// TIA Portal V15.1 export
// export: Created 2024-05-17T05:38:09.4997729Z, ExportSetting WithDefaults, DisplayName Totally Integrated Automation Portal, DisplayVersion V15.1 Update 5, DisplayName TIA Portal Openness, DisplayVersion V15.1 Update 5, DisplayName SINAMICS Startdrive Advanced, DisplayVersion V15.1, DisplayName G130, G150, S120, S150, SINAMICS MV, S210, DisplayVersion V15.1, DisplayName G110M, G120, G120C, G120D, G120P, DisplayVersion V15.1, DisplayName STEP 7 Professional, DisplayVersion V15.1 Update 5, DisplayName STEP 7 Safety, DisplayVersion V15.1, DisplayName WinCC Professional, DisplayVersion V15.1 Update 5, DisplayName SIMATIC Visualization Architect, DisplayVersion V15.1
ORGANIZATION_BLOCK "209000NCP01"   // OB1, FBD, ProgramCycle
TITLE = 209000NCP01
{ S7_Optimized_Access := 'FALSE' }
VERSION : 0.1
// stored: AutoNumber false, IsIECCheckEnabled false, SetENOAutomatically False
   VAR_TEMP
      OB1_EV_CLASS : Byte;   // Bits 0-3 = 1 (Coming event), Bits 4-7 = 1 (Event class 1)
      OB1_SCAN_1 : Byte;   // 1 (Cold restart scan 1 of OB 1), 3 (Scan 2-n of OB 1)
      OB1_PRIORITY : Byte;   // Priority of OB Execution
      OB1_OB_NUMBR : Byte;   // 1 (Organization block 1, OB1)
      OB1_RESERVED_1 : Byte;   // Reserved for system
      OB1_RESERVED_2 : Byte;   // Reserved for system
      OB1_PREV_CYCLE : Int;   // Cycle time of previous OB1 scan (milliseconds)
      OB1_MIN_CYCLE : Int;   // Minimum cycle time of OB1 (milliseconds)
      OB1_MAX_CYCLE : Int;   // Maximum cycle time of OB1 (milliseconds)
      OB1_DATE_TIME : Date_And_Time;   // Date and time OB1 started
   END_VAR
BEGIN

REGION Network 1: **** 1 - Inputs **** Incrementation of number of executions
   // Incrementation of number of executions
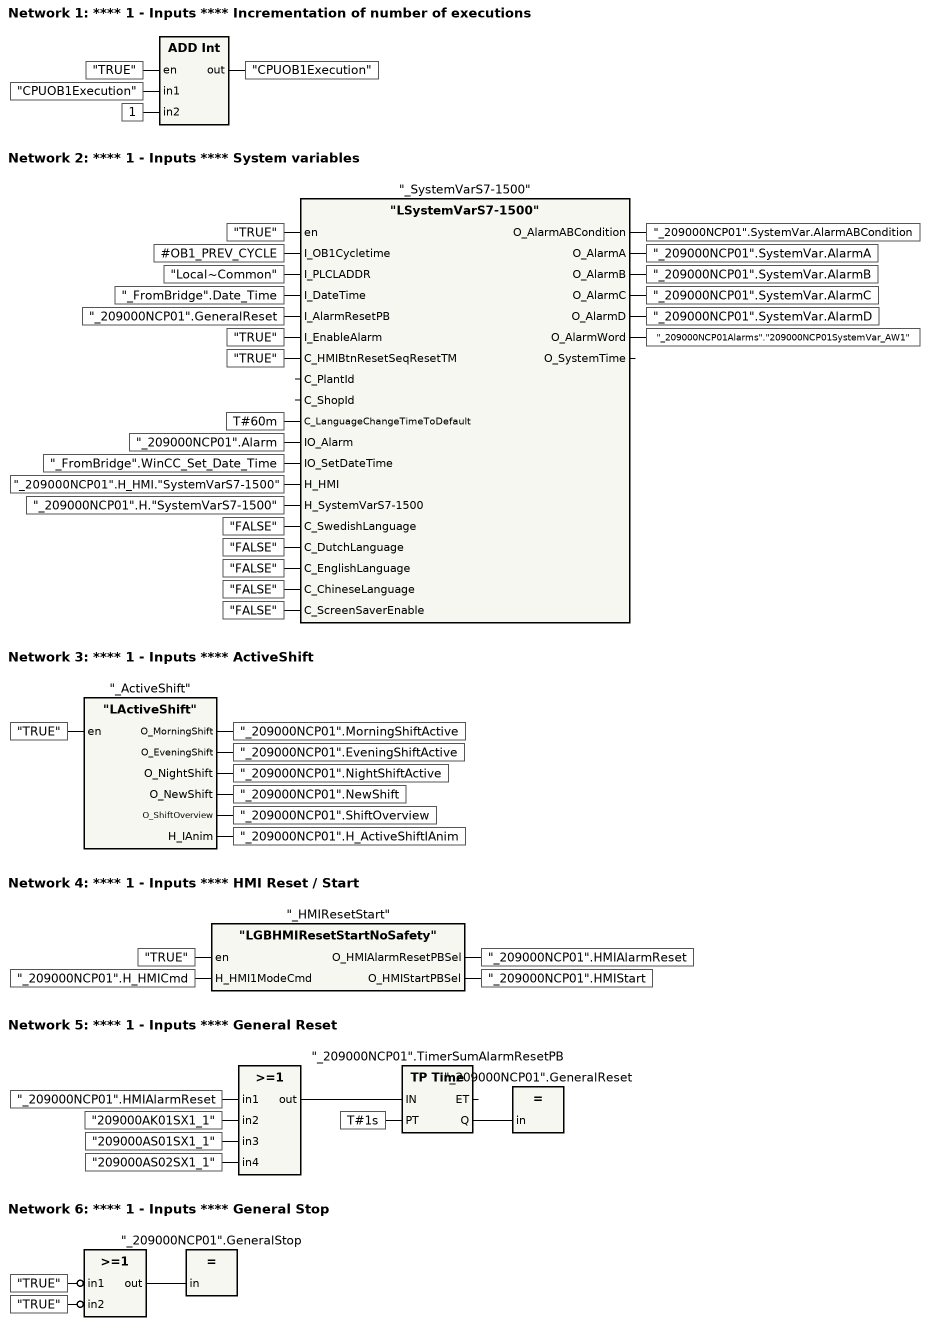
   IF "TRUE" THEN "CPUOB1Execution" := "CPUOB1Execution" + 1; END_IF;
END_REGION

REGION Network 2: **** 1 - Inputs **** System variables
   // System variables
   IF "TRUE" THEN
       "_SystemVarS7-1500"(I_OB1Cycletime := #OB1_PREV_CYCLE,   // "LSystemVarS7-1500"
                           I_PLCLADDR := "Local~Common",
                           I_DateTime := "_FromBridge".Date_Time,
                           I_AlarmResetPB := "_209000NCP01".GeneralReset,
                           I_EnableAlarm := "TRUE",
                           C_HMIBtnResetSeqResetTM := "TRUE",
                           C_LanguageChangeTimeToDefault := T#60m,
                           IO_Alarm := "_209000NCP01".Alarm,
                           IO_SetDateTime := "_FromBridge".WinCC_Set_Date_Time,
                           H_HMI := "_209000NCP01".H_HMI."SystemVarS7-1500",
                           "H_SystemVarS7-1500" := "_209000NCP01".H."SystemVarS7-1500",
                           C_SwedishLanguage := "FALSE",
                           C_DutchLanguage := "FALSE",
                           C_EnglishLanguage := "FALSE",
                           C_ChineseLanguage := "FALSE",
                           C_ScreenSaverEnable := "FALSE",
                           O_AlarmABCondition => "_209000NCP01".SystemVar.AlarmABCondition,
                           O_AlarmA => "_209000NCP01".SystemVar.AlarmA,
                           O_AlarmB => "_209000NCP01".SystemVar.AlarmB,
                           O_AlarmC => "_209000NCP01".SystemVar.AlarmC,
                           O_AlarmD => "_209000NCP01".SystemVar.AlarmD,
                           O_AlarmWord => "_209000NCP01Alarms"."209000NCP01SystemVar_AW1");
   END_IF;
END_REGION

REGION Network 3: **** 1 - Inputs **** ActiveShift
   // ActiveShift
   IF "TRUE" THEN
       "_ActiveShift"(O_MorningShift => "_209000NCP01".MorningShiftActive,   // "LActiveShift"
                      O_EveningShift => "_209000NCP01".EveningShiftActive,
                      O_NightShift => "_209000NCP01".NightShiftActive,
                      O_NewShift => "_209000NCP01".NewShift,
                      O_ShiftOverview => "_209000NCP01".ShiftOverview,
                      H_IAnim => "_209000NCP01".H_ActiveShiftIAnim);
   END_IF;
END_REGION

REGION Network 4: **** 1 - Inputs **** HMI Reset / Start
   // Alarm reset and Start from Main picture
   // Note: connect signal "Safety not ok" from the failsafe program
   IF "TRUE" THEN
       "_HMIResetStart"(H_HMI1ModeCmd := "_209000NCP01".H_HMICmd,   // "LGBHMIResetStartNoSafety"
                        O_HMIAlarmResetPBSel => "_209000NCP01".HMIAlarmReset,
                        O_HMIStartPBSel => "_209000NCP01".HMIStart);
   END_IF;
END_REGION

REGION Network 5: **** 1 - Inputs **** General Reset
   // Alarm reset pushbuttons
   // Note: Add all the hardware buttons for general alarm reset
   "_209000NCP01".TimerSumAlarmResetPB.TP(IN := "_209000NCP01".HMIAlarmReset OR "209000AK01SX1_1" OR "209000AS01SX1_1" OR "209000AS02SX1_1",
                           PT := T#1s);
   "_209000NCP01".GeneralReset := "_209000NCP01".TimerSumAlarmResetPB.Q;
END_REGION

REGION Network 6: **** 1 - Inputs **** General Stop
   // Stop pushbuttons
   // Note: Add all the hardware buttons for general stop
   "_209000NCP01".GeneralStop := NOT "TRUE" OR NOT "TRUE";
END_REGION

REGION Network 7: **** 1 - Inputs **** Summary of all start buttons
   // Summation of all Start pushbuttons
   // Note: Add all the hardware buttons for general start
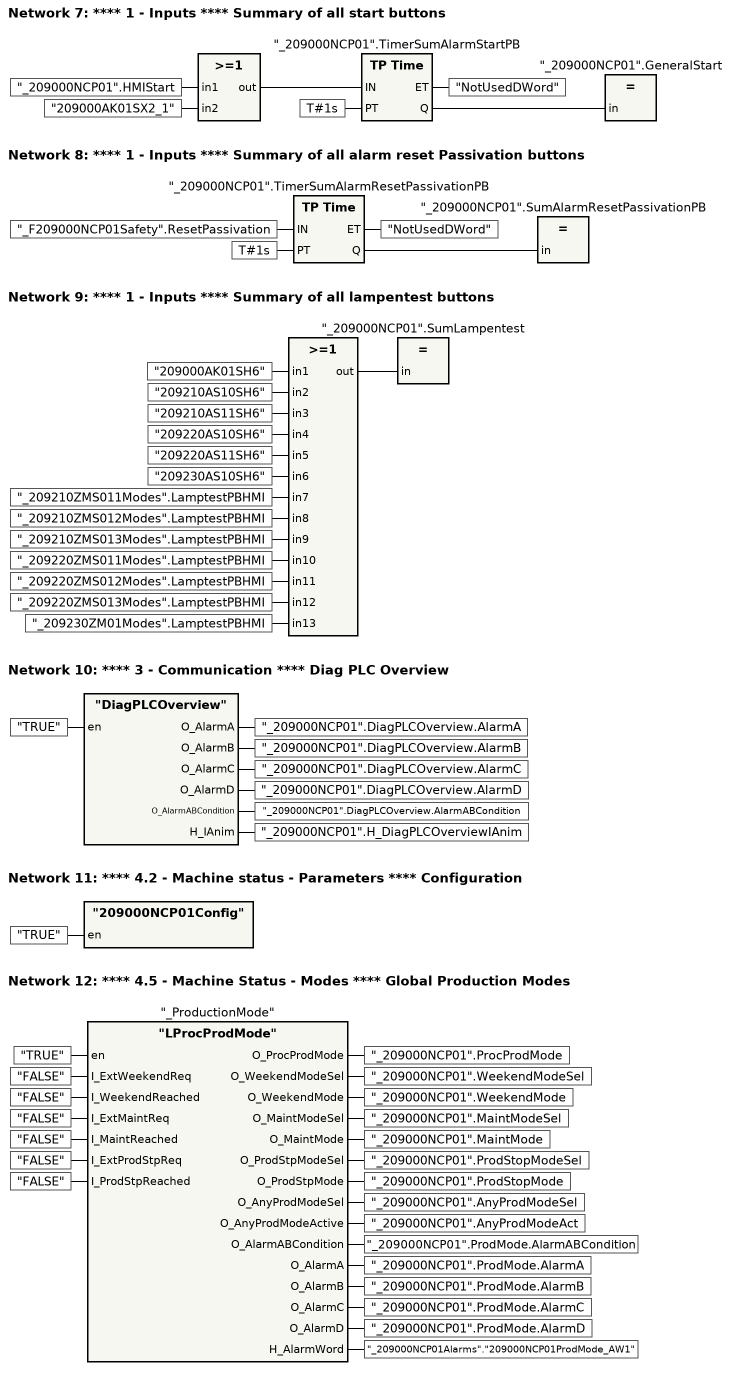
   "_209000NCP01".TimerSumAlarmStartPB.TP(IN := "_209000NCP01".HMIStart OR "209000AK01SX2_1",
                           PT := T#1s,
                           ET => "NotUsedDWord");
   "_209000NCP01".GeneralStart := "_209000NCP01".TimerSumAlarmStartPB.Q;
END_REGION

REGION Network 8: **** 1 - Inputs **** Summary of all alarm reset Passivation buttons
   // Summary of all alarm reset Passivation buttons
   "_209000NCP01".TimerSumAlarmResetPassivationPB.TP(IN := "_F209000NCP01Safety".ResetPassivation,
                           PT := T#1s,
                           ET => "NotUsedDWord");
   "_209000NCP01".SumAlarmResetPassivationPB := "_209000NCP01".TimerSumAlarmResetPassivationPB.Q;
END_REGION

REGION Network 9: **** 1 - Inputs **** Summary of all lampentest buttons
   "_209000NCP01".SumLampentest := "209000AK01SH6" OR "209210AS10SH6" OR "209210AS11SH6" OR "209220AS10SH6" OR "209220AS11SH6" OR "209230AS10SH6" OR "_209210ZMS011Modes".LamptestPBHMI OR "_209210ZMS012Modes".LamptestPBHMI OR "_209210ZMS013Modes".LamptestPBHMI OR "_209220ZMS011Modes".LamptestPBHMI OR "_209220ZMS012Modes".LamptestPBHMI OR "_209220ZMS013Modes".LamptestPBHMI OR "_209230ZM01Modes".LamptestPBHMI;
END_REGION

REGION Network 10: **** 3 - Communication **** Diag PLC Overview
   // PLC items
   // Safety, Profibus
   IF "TRUE" THEN
       "DiagPLCOverview"(O_AlarmA => "_209000NCP01".DiagPLCOverview.AlarmA,
                         O_AlarmB => "_209000NCP01".DiagPLCOverview.AlarmB,
                         O_AlarmC => "_209000NCP01".DiagPLCOverview.AlarmC,
                         O_AlarmD => "_209000NCP01".DiagPLCOverview.AlarmD,
                         O_AlarmABCondition => "_209000NCP01".DiagPLCOverview.AlarmABCondition,
                         H_IAnim => "_209000NCP01".H_DiagPLCOverviewIAnim);
   END_IF;
END_REGION

REGION Network 11: **** 4.2 - Machine status - Parameters **** Configuration
   IF "TRUE" THEN "209000NCP01Config"(); END_IF;
END_REGION

REGION Network 12: **** 4.5 - Machine Status - Modes **** Global Production Modes
   // Global Production Modes
   IF "TRUE" THEN
       "_ProductionMode"(I_ExtWeekendReq := "FALSE",   // "LProcProdMode"
                         I_WeekendReached := "FALSE",
                         I_ExtMaintReq := "FALSE",
                         I_MaintReached := "FALSE",
                         I_ExtProdStpReq := "FALSE",
                         I_ProdStpReached := "FALSE",
                         O_ProcProdMode => "_209000NCP01".ProcProdMode,
                         O_WeekendModeSel => "_209000NCP01".WeekendModeSel,
                         O_WeekendMode => "_209000NCP01".WeekendMode,
                         O_MaintModeSel => "_209000NCP01".MaintModeSel,
                         O_MaintMode => "_209000NCP01".MaintMode,
                         O_ProdStpModeSel => "_209000NCP01".ProdStopModeSel,
                         O_ProdStpMode => "_209000NCP01".ProdStopMode,
                         O_AnyProdModeSel => "_209000NCP01".AnyProdModeSel,
                         O_AnyProdModeActive => "_209000NCP01".AnyProdModeAct,
                         O_AlarmABCondition => "_209000NCP01".ProdMode.AlarmABCondition,
                         O_AlarmA => "_209000NCP01".ProdMode.AlarmA,
                         O_AlarmB => "_209000NCP01".ProdMode.AlarmB,
                         O_AlarmC => "_209000NCP01".ProdMode.AlarmC,
                         O_AlarmD => "_209000NCP01".ProdMode.AlarmD,
                         H_AlarmWord => "_209000NCP01Alarms"."209000NCP01ProdMode_AW1");
   END_IF;
END_REGION

REGION Network 13: **** 4.5 - Machine Status - Modes **** Global Production Modes
   // Global Production Modes
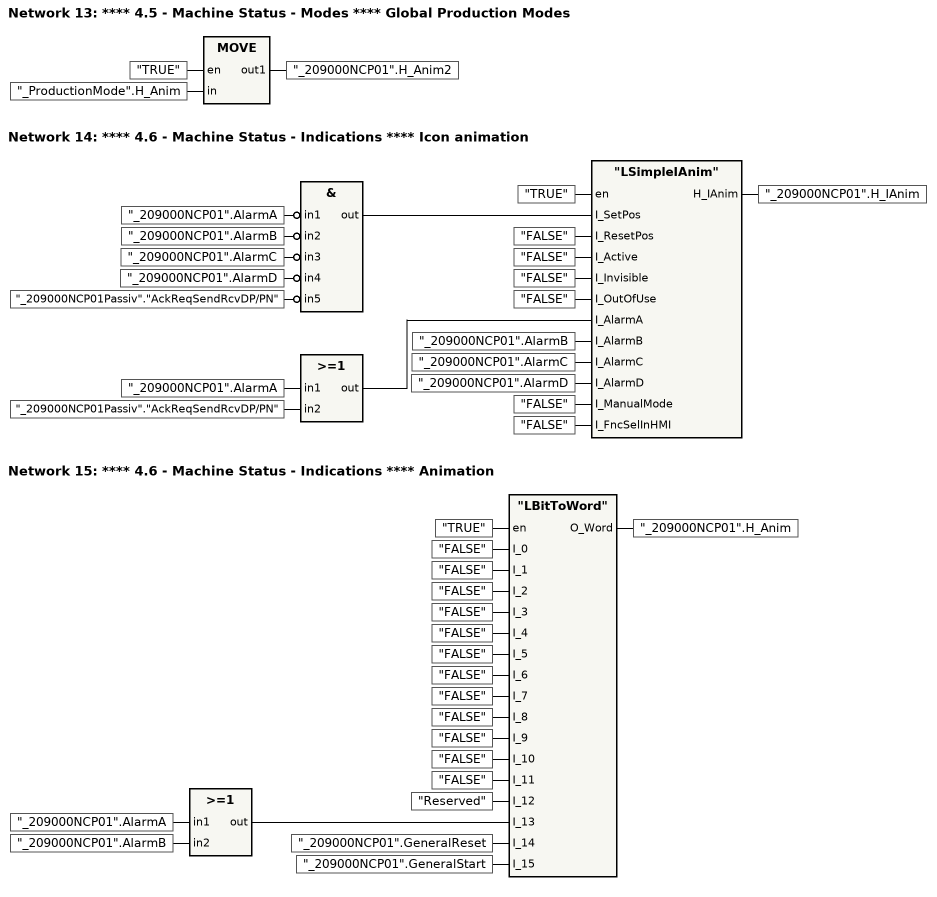
   IF "TRUE" THEN "_209000NCP01".H_Anim2 := "_ProductionMode".H_Anim; END_IF;
END_REGION

REGION Network 14: **** 4.6 - Machine Status - Indications **** Icon animation
   // Icon animation
   IF "TRUE" THEN
       "LSimpleIAnim"(I_SetPos := NOT "_209000NCP01".AlarmA AND NOT "_209000NCP01".AlarmB AND NOT "_209000NCP01".AlarmC AND NOT "_209000NCP01".AlarmD AND NOT "_209000NCP01Passiv"."AckReqSendRcvDP/PN",
                      I_ResetPos := "FALSE",
                      I_Active := "FALSE",
                      I_Invisible := "FALSE",
                      I_OutOfUse := "FALSE",
                      I_AlarmA := "_209000NCP01".AlarmA OR "_209000NCP01Passiv"."AckReqSendRcvDP/PN",
                      I_AlarmB := "_209000NCP01".AlarmB,
                      I_AlarmC := "_209000NCP01".AlarmC,
                      I_AlarmD := "_209000NCP01".AlarmD,
                      I_ManualMode := "FALSE",
                      I_FncSelInHMI := "FALSE",
                      H_IAnim => "_209000NCP01".H_IAnim);
   END_IF;
END_REGION

REGION Network 15: **** 4.6 - Machine Status - Indications **** Animation
   // Animation
   // Note: Bit 10 = Alarm reset button HMI
   //       Bit 12 = SafetyResetable (shows popup ACK SAFETY when this bit is set)
   //       Bit 15 = Any Upperlevel A or B alarm
   IF "TRUE" THEN
       "LBitToWord"(I_0 := "FALSE",
                    I_1 := "FALSE",
                    I_2 := "FALSE",
                    I_3 := "FALSE",
                    I_4 := "FALSE",
                    I_5 := "FALSE",
                    I_6 := "FALSE",
                    I_7 := "FALSE",
                    I_8 := "FALSE",
                    I_9 := "FALSE",
                    I_10 := "FALSE",
                    I_11 := "FALSE",
                    I_12 := "Reserved",
                    I_13 := "_209000NCP01".AlarmA OR "_209000NCP01".AlarmB,
                    I_14 := "_209000NCP01".GeneralReset,
                    I_15 := "_209000NCP01".GeneralStart,
                    O_Word => "_209000NCP01".H_Anim);
   END_IF;
END_REGION

NETWORK
TITLE = **** 4.6 - Machine Status - Indications **** Animation DB number
// DB number
      OPN   "_209000NCP01";
      L     DBNO;
      T     "_209000NCP01".H_DBnr;

REGION Network 17: **** 4.6 - Machine Status - Indication **** LED Indication 209000AK01 - Start/Reset
   // This module handles indication for Start and Reset buttons on AK01
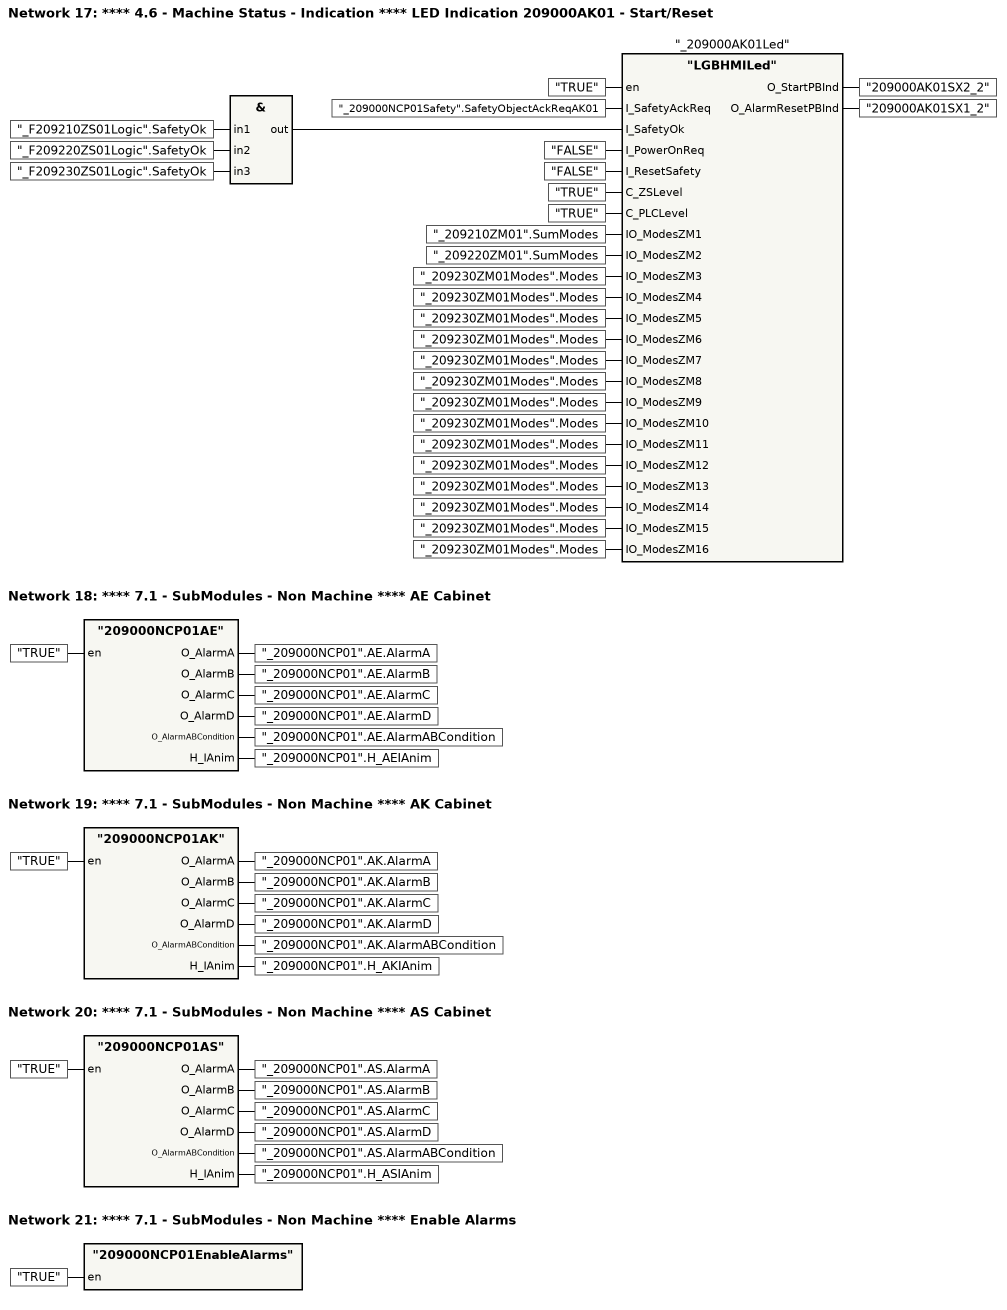
   IF "TRUE" THEN
       "_209000AK01Led"(I_SafetyAckReq := "_209000NCP01Safety".SafetyObjectAckReqAK01,   // "LGBHMILed"
                        I_SafetyOk := "_F209210ZS01Logic".SafetyOk AND "_F209220ZS01Logic".SafetyOk AND "_F209230ZS01Logic".SafetyOk,
                        I_PowerOnReq := "FALSE",
                        I_ResetSafety := "FALSE",
                        C_ZSLevel := "TRUE",
                        C_PLCLevel := "TRUE",
                        IO_ModesZM1 := "_209210ZM01".SumModes,
                        IO_ModesZM2 := "_209220ZM01".SumModes,
                        IO_ModesZM3 := "_209230ZM01Modes".Modes,
                        IO_ModesZM4 := "_209230ZM01Modes".Modes,
                        IO_ModesZM5 := "_209230ZM01Modes".Modes,
                        IO_ModesZM6 := "_209230ZM01Modes".Modes,
                        IO_ModesZM7 := "_209230ZM01Modes".Modes,
                        IO_ModesZM8 := "_209230ZM01Modes".Modes,
                        IO_ModesZM9 := "_209230ZM01Modes".Modes,
                        IO_ModesZM10 := "_209230ZM01Modes".Modes,
                        IO_ModesZM11 := "_209230ZM01Modes".Modes,
                        IO_ModesZM12 := "_209230ZM01Modes".Modes,
                        IO_ModesZM13 := "_209230ZM01Modes".Modes,
                        IO_ModesZM14 := "_209230ZM01Modes".Modes,
                        IO_ModesZM15 := "_209230ZM01Modes".Modes,
                        IO_ModesZM16 := "_209230ZM01Modes".Modes,
                        O_StartPBInd => "209000AK01SX2_2",
                        O_AlarmResetPBInd => "209000AK01SX1_2");
   END_IF;
END_REGION

REGION Network 18: **** 7.1 - SubModules - Non Machine **** AE Cabinet
   // AE Cabinet
   IF "TRUE" THEN
       "209000NCP01AE"(O_AlarmA => "_209000NCP01".AE.AlarmA,
                       O_AlarmB => "_209000NCP01".AE.AlarmB,
                       O_AlarmC => "_209000NCP01".AE.AlarmC,
                       O_AlarmD => "_209000NCP01".AE.AlarmD,
                       O_AlarmABCondition => "_209000NCP01".AE.AlarmABCondition,
                       H_IAnim => "_209000NCP01".H_AEIAnim);
   END_IF;
END_REGION

REGION Network 19: **** 7.1 - SubModules - Non Machine **** AK Cabinet
   // AK cabinet
   IF "TRUE" THEN
       "209000NCP01AK"(O_AlarmA => "_209000NCP01".AK.AlarmA,
                       O_AlarmB => "_209000NCP01".AK.AlarmB,
                       O_AlarmC => "_209000NCP01".AK.AlarmC,
                       O_AlarmD => "_209000NCP01".AK.AlarmD,
                       O_AlarmABCondition => "_209000NCP01".AK.AlarmABCondition,
                       H_IAnim => "_209000NCP01".H_AKIAnim);
   END_IF;
END_REGION

REGION Network 20: **** 7.1 - SubModules - Non Machine **** AS Cabinet
   // AS Cabinet Alarms
   IF "TRUE" THEN
       "209000NCP01AS"(O_AlarmA => "_209000NCP01".AS.AlarmA,
                       O_AlarmB => "_209000NCP01".AS.AlarmB,
                       O_AlarmC => "_209000NCP01".AS.AlarmC,
                       O_AlarmD => "_209000NCP01".AS.AlarmD,
                       O_AlarmABCondition => "_209000NCP01".AS.AlarmABCondition,
                       H_IAnim => "_209000NCP01".H_ASIAnim);
   END_IF;
END_REGION

REGION Network 21: **** 7.1 - SubModules - Non Machine **** Enable Alarms
   IF "TRUE" THEN "209000NCP01EnableAlarms"(); END_IF;
END_REGION

REGION Network 22: **** 7.1 - Submodule - Non Machine **** Safety <-> Non Safety
   // Signals between safety program and non safety program
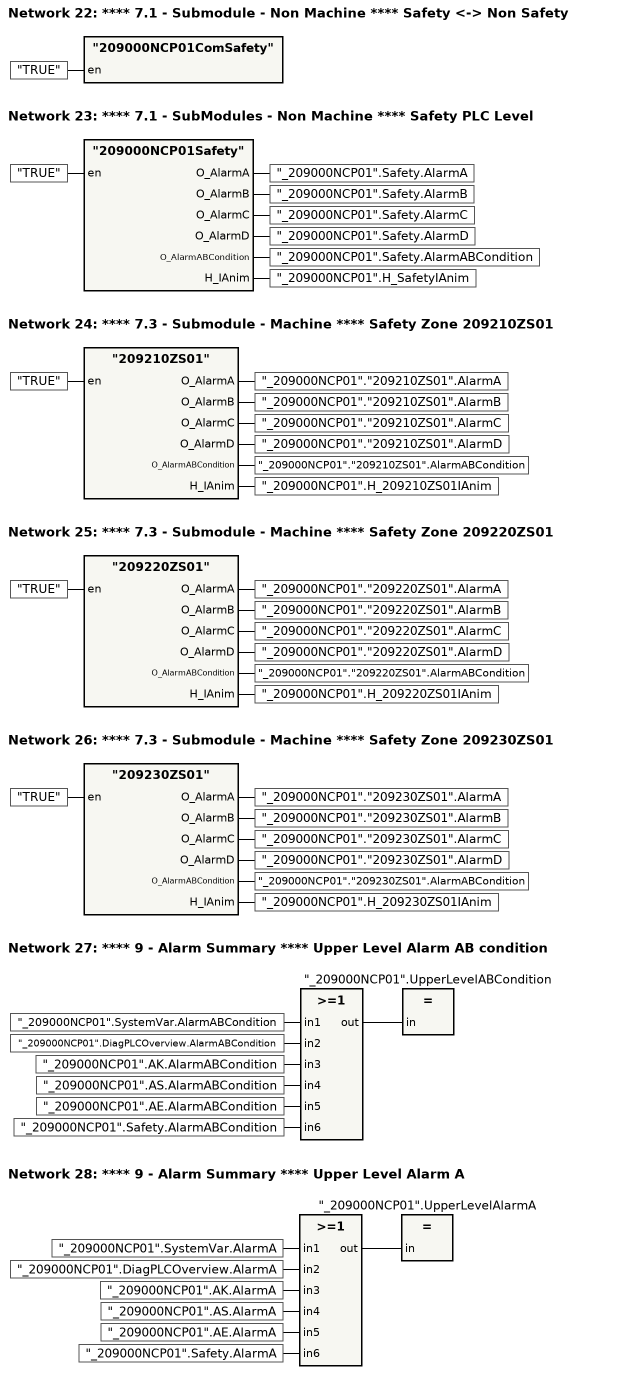
   IF "TRUE" THEN "209000NCP01ComSafety"(); END_IF;
END_REGION

REGION Network 23: **** 7.1 - SubModules - Non Machine **** Safety PLC Level
   // General Safety on PLC Level
   IF "TRUE" THEN
       "209000NCP01Safety"(O_AlarmA => "_209000NCP01".Safety.AlarmA,
                           O_AlarmB => "_209000NCP01".Safety.AlarmB,
                           O_AlarmC => "_209000NCP01".Safety.AlarmC,
                           O_AlarmD => "_209000NCP01".Safety.AlarmD,
                           O_AlarmABCondition => "_209000NCP01".Safety.AlarmABCondition,
                           H_IAnim => "_209000NCP01".H_SafetyIAnim);
   END_IF;
END_REGION

REGION Network 24: **** 7.3 - Submodule - Machine **** Safety Zone 209210ZS01
   // Safety Zone
   IF "TRUE" THEN
       "209210ZS01"(O_AlarmA => "_209000NCP01"."209210ZS01".AlarmA,
                    O_AlarmB => "_209000NCP01"."209210ZS01".AlarmB,
                    O_AlarmC => "_209000NCP01"."209210ZS01".AlarmC,
                    O_AlarmD => "_209000NCP01"."209210ZS01".AlarmD,
                    O_AlarmABCondition => "_209000NCP01"."209210ZS01".AlarmABCondition,
                    H_IAnim => "_209000NCP01".H_209210ZS01IAnim);
   END_IF;
END_REGION

REGION Network 25: **** 7.3 - Submodule - Machine **** Safety Zone 209220ZS01
   // Safety Zone
   IF "TRUE" THEN
       "209220ZS01"(O_AlarmA => "_209000NCP01"."209220ZS01".AlarmA,
                    O_AlarmB => "_209000NCP01"."209220ZS01".AlarmB,
                    O_AlarmC => "_209000NCP01"."209220ZS01".AlarmC,
                    O_AlarmD => "_209000NCP01"."209220ZS01".AlarmD,
                    O_AlarmABCondition => "_209000NCP01"."209220ZS01".AlarmABCondition,
                    H_IAnim => "_209000NCP01".H_209220ZS01IAnim);
   END_IF;
END_REGION

REGION Network 26: **** 7.3 - Submodule - Machine **** Safety Zone 209230ZS01
   // Safety Zone
   IF "TRUE" THEN
       "209230ZS01"(O_AlarmA => "_209000NCP01"."209230ZS01".AlarmA,
                    O_AlarmB => "_209000NCP01"."209230ZS01".AlarmB,
                    O_AlarmC => "_209000NCP01"."209230ZS01".AlarmC,
                    O_AlarmD => "_209000NCP01"."209230ZS01".AlarmD,
                    O_AlarmABCondition => "_209000NCP01"."209230ZS01".AlarmABCondition,
                    H_IAnim => "_209000NCP01".H_209230ZS01IAnim);
   END_IF;
END_REGION

REGION Network 27: **** 9 - Alarm Summary **** Upper Level Alarm AB condition
   // UpperLevel Alarm AB condition
   "_209000NCP01".UpperLevelABCondition := "_209000NCP01".SystemVar.AlarmABCondition OR "_209000NCP01".DiagPLCOverview.AlarmABCondition OR "_209000NCP01".AK.AlarmABCondition OR "_209000NCP01".AS.AlarmABCondition OR "_209000NCP01".AE.AlarmABCondition OR "_209000NCP01".Safety.AlarmABCondition;
END_REGION

REGION Network 28: **** 9 - Alarm Summary **** Upper Level Alarm A
   // UpperLevel AlarmA for lower level application (modezone)
   // Note: Connect all AlarmA which are to be sent to the lower level
   "_209000NCP01".UpperLevelAlarmA := "_209000NCP01".SystemVar.AlarmA OR "_209000NCP01".DiagPLCOverview.AlarmA OR "_209000NCP01".AK.AlarmA OR "_209000NCP01".AS.AlarmA OR "_209000NCP01".AE.AlarmA OR "_209000NCP01".Safety.AlarmA;
END_REGION

REGION Network 29: **** 9 - Alarm Summary **** Upper Level Alarm B
   // UpperLevelAlarmB for lower level application (modezone)
   // Note: Connect all AlarmB which are to be sent to the lower level
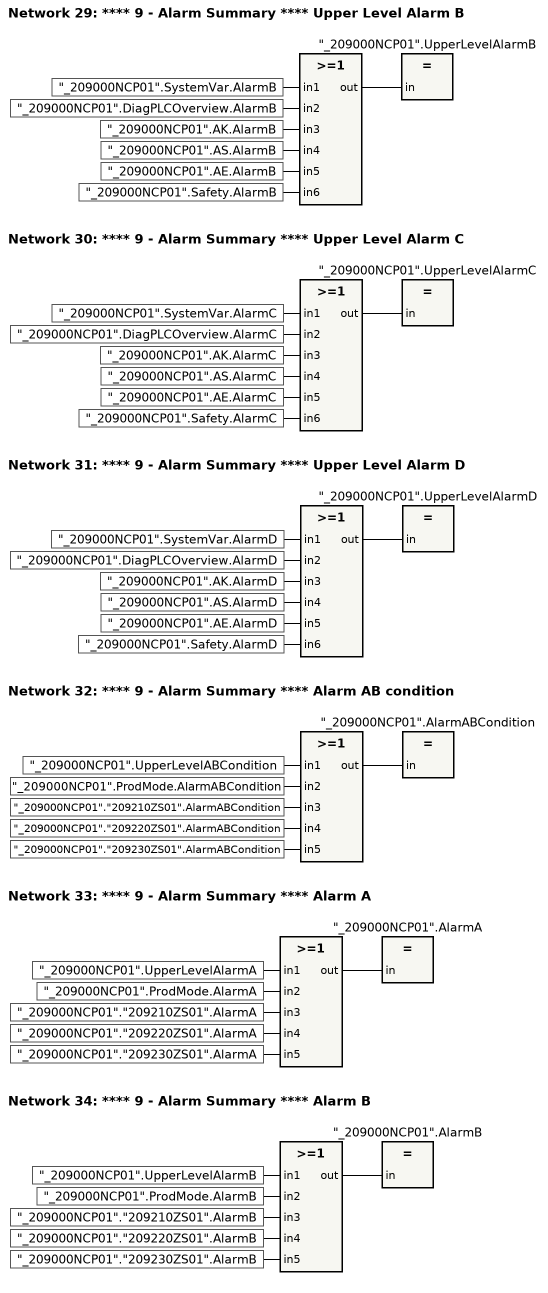
   "_209000NCP01".UpperLevelAlarmB := "_209000NCP01".SystemVar.AlarmB OR "_209000NCP01".DiagPLCOverview.AlarmB OR "_209000NCP01".AK.AlarmB OR "_209000NCP01".AS.AlarmB OR "_209000NCP01".AE.AlarmB OR "_209000NCP01".Safety.AlarmB;
END_REGION

REGION Network 30: **** 9 - Alarm Summary **** Upper Level Alarm C
   // UpperLevelAlarmC for lower level application (modezone)
   // Note: Connect all AlarmC which are to be sent to the lower level
   "_209000NCP01".UpperLevelAlarmC := "_209000NCP01".SystemVar.AlarmC OR "_209000NCP01".DiagPLCOverview.AlarmC OR "_209000NCP01".AK.AlarmC OR "_209000NCP01".AS.AlarmC OR "_209000NCP01".AE.AlarmC OR "_209000NCP01".Safety.AlarmC;
END_REGION

REGION Network 31: **** 9 - Alarm Summary **** Upper Level Alarm D
   // UpperLevelAlarmD for lower level application (modezone)
   // Note: Connect all AlarmD which are to be sent to the lower level
   "_209000NCP01".UpperLevelAlarmD := "_209000NCP01".SystemVar.AlarmD OR "_209000NCP01".DiagPLCOverview.AlarmD OR "_209000NCP01".AK.AlarmD OR "_209000NCP01".AS.AlarmD OR "_209000NCP01".AE.AlarmD OR "_209000NCP01".Safety.AlarmD;
END_REGION

REGION Network 32: **** 9 - Alarm Summary **** Alarm AB condition
   // Alarm AB condition
   "_209000NCP01".AlarmABCondition := "_209000NCP01".UpperLevelABCondition OR "_209000NCP01".ProdMode.AlarmABCondition OR "_209000NCP01"."209210ZS01".AlarmABCondition OR "_209000NCP01"."209220ZS01".AlarmABCondition OR "_209000NCP01"."209230ZS01".AlarmABCondition;
END_REGION

REGION Network 33: **** 9 - Alarm Summary **** Alarm A
   // Alarm A
   "_209000NCP01".AlarmA := "_209000NCP01".UpperLevelAlarmA OR "_209000NCP01".ProdMode.AlarmA OR "_209000NCP01"."209210ZS01".AlarmA OR "_209000NCP01"."209220ZS01".AlarmA OR "_209000NCP01"."209230ZS01".AlarmA;
END_REGION

REGION Network 34: **** 9 - Alarm Summary **** Alarm B
   // Alarm B
   "_209000NCP01".AlarmB := "_209000NCP01".UpperLevelAlarmB OR "_209000NCP01".ProdMode.AlarmB OR "_209000NCP01"."209210ZS01".AlarmB OR "_209000NCP01"."209220ZS01".AlarmB OR "_209000NCP01"."209230ZS01".AlarmB;
END_REGION

REGION Network 35: **** 9 - Alarm Summary **** Alarm C
   // Alarm C
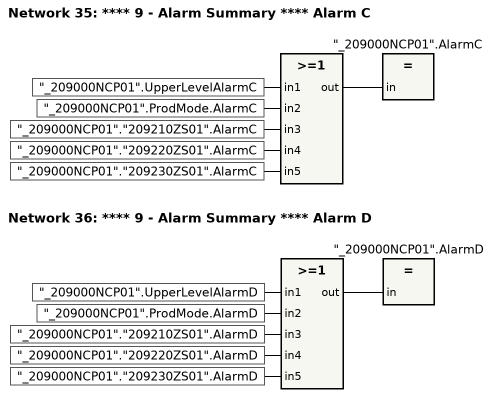
   "_209000NCP01".AlarmC := "_209000NCP01".UpperLevelAlarmC OR "_209000NCP01".ProdMode.AlarmC OR "_209000NCP01"."209210ZS01".AlarmC OR "_209000NCP01"."209220ZS01".AlarmC OR "_209000NCP01"."209230ZS01".AlarmC;
END_REGION

REGION Network 36: **** 9 - Alarm Summary **** Alarm D
   // Alarm D
   "_209000NCP01".AlarmD := "_209000NCP01".UpperLevelAlarmD OR "_209000NCP01".ProdMode.AlarmD OR "_209000NCP01"."209210ZS01".AlarmD OR "_209000NCP01"."209220ZS01".AlarmD OR "_209000NCP01"."209230ZS01".AlarmD;
END_REGION
END_ORGANIZATION_BLOCK
